{attribute 'qualified_only'}
{attribute 'strict'}
TYPE E_LCLSMotionError :
(
    ABORTED := 16#7900,
    UNSAFE := 16#7901,
    INVALID := 16#7902,
    MCS2_FAULT := 16#7903,
    TEST := 16#FFFF
) UDINT;
END_TYPE

(* stored: Version 1.1.0.1
   DUT E_LCLSMotionError: Id {ddea4357-8fae-44da-b5b7-bd2ca001f059} *)
